TEXTLIST TextList_EcoMode
  0 = 'Activation Eco-veille' | FR: 'Activation Eco-veille' | EN: 'Eco-sleep activation'
  1 = 'Temps inav' | FR: "Temps d'inactivité avant Eco-veille" | EN: 'Inactivity time before eco-sleep'
  2 = 'Process deep eco-sleep' | FR: 'Procédé Eco-veille profond' | EN: 'Deep eco-sleep process'
  3 = 'Record' | FR: 'Enregistrement' | EN: 'Record'
  4 = 'Select' | FR: '...' | EN: '...'
  5 = 'Canon actif' | FR: 'Evap. active' | EN: 'Evap. on'
  6 = 'On/Off' | FR: 'Activation/Désactivation' | EN: 'On/Off'
  7 = 'Evap On/Off' | FR: 'Activation/Désactivation Evap.' | EN: 'Evap. On/Off'
  8 = 'Eco Mode' | FR: 'Eco-veille' | EN: 'Eco-sleep'
  9 = 'Config' | FR: 'Configuration' | EN: 'Configuration'
  10 = 'Eco Mode actif' | FR: 'Eco-veille actif' | EN: 'Eco-sleep On'
  11 = 'Inactivité' | FR: 'Inactivité :' | EN: 'Inactivity :'
  12 = " Lancement du procédé eco-veille profond à l'issue de la production" | FR: " Lancement du procédé Eco-veille profond à l'issue de la production" | EN: 'Start the deep eco-sleep process at the end of the production'
   = ''
END_TEXTLIST

(* stored: Version 1.1.0.1, ProductVersion 3.1.4024.10
   TextList TextList_EcoMode: Id {4e113988-9321-43c0-8b72-edce0f3adacc} *)
